TYPE ST_ProtectionSystems_get :
STRUCT
	//Fire Detection System
	FireDetection						: REFERENCE TO ST_Firedetection_get;
	
	//InsulationMonitor
	Insulation							: REFERENCE TO ST_InsulationMonitor_get;
	
	//MRCDB
	MRCDB								: REFERENCE TO ST_ResidualCurrentMonitor_get;
	
	//Surge protection
	Surge								: REFERENCE TO ST_SurgeProtection_get;
	
	//Overcurrent protection
	OvercurrentProtection				: REFERENCE TO ST_OverCurrentProtection_Get;
	
END_STRUCT
END_TYPE

(* stored: Version 1.1.0.1, ProductVersion 3.1.4024.12
   DUT ST_ProtectionSystems_get: Id {c1c9b2be-98af-477c-aa1b-0263e2a01a7a} *)
